{attribute 'qualified_only'}
TYPE E_LogicOperator :
(
	LOGIC_OP_UNDEFINED := 0,
	LOGIC_OP_AND := 1,
	LOGIC_OP_OR := 2
)USINT;
END_TYPE

(* stored: Version 1.1.0.1, ProductVersion 3.1.4020.12
   DUT E_LogicOperator: Id {cfd2b225-520a-4908-a170-625490dabc77} *)
